FUNCTION_BLOCK FB_MachineController
VAR
	iConveyer : I_Conveyer;
	ePreviousMachineState : E_MachineState;
	fbTimer : TON;
	tWaitTime : TIME := T#10S;
	tProcessTime : TIME := T#5S;
	fbAutoTimer : TON;
END_VAR

IF GVL_HMI.bStop THEN
	IF GVL_HMI.eMachineState =  E_MachineState.STOPPED THEN
		GVL_HMI.eMachineState := E_MachineState.IDLE;
	ELSE
		ePreviousMachineState := GVL_HMI.eMachineState ;
		GVL_HMI.eMachineState := E_MachineState.STOPPED;
	END_IF
	fbTimer(IN := FALSE, PT := tWaitTime);
	GVL_HMI.bStop := FALSE;
	
END_IF
CASE GVL_HMI.eMachineState OF
	E_MachineState.IDLE :
		IF GVL_HMI.bStart THEN
			GVL_HMI.bStart := FALSE;
			IF iConveyer <> 0 THEN
					ePreviousMachineState := GVL_HMI.eMachineState ;
					GVL_HMI.eMachineState := E_MachineState.WAIT_FOR_BOTTLE;
			ELSE
				ePreviousMachineState := GVL_HMI.eMachineState ;
				GVL_HMI.eMachineState := E_MachineState.ERROR;
			END_IF
		END_IF
		
	E_MachineState.WAIT_FOR_BOTTLE :
		iConveyer.Start();
		fbTimer ( IN:= TRUE, PT:= tWaitTime);
		IF fbTimer.Q THEN
			fbTimer(IN := FALSE);
			GVL_HMI.eAlarmState := E_AlarmState.BOTTLE_SENSOR;
			GVL_HMI.eMachineState := E_MachineState.ERROR;
		END_IF
		//AutoMode
		IF GVL_HMI.eMachineMode = E_MachineMode.Auto THEN
			fbAutoTimer(IN := TRUE, PT := tProcessTime);
			IF fbAutoTimer.Q THEN
				fbAutoTimer(IN := FALSE);
				GVL_HMI.bBottleSensor := TRUE;
			END_IF
		ELSE
			fbAutoTimer(IN := FALSE);
		END_IF
		
		IF GVL_HMI.bBottleSensor THEN
				GVL_HMI.bBottleSensor := FALSE;
				fbTimer(IN := FALSE);
				iConveyer.Stop();
				ePreviousMachineState := GVL_HMI.eMachineState ;
				GVL_HMI.eMachineState := E_MachineState.FILLING;
		END_IF
	
	E_MachineState.FILLING :
		GVL_HMI.bFillingValve := TRUE;
		fbTimer ( IN:= TRUE, PT:= tWaitTime);
		IF fbTimer.Q THEN
			fbTimer(IN := FALSE);
			GVL_HMI.eAlarmState := E_AlarmState.LEVEL_SENSOR;
			GVL_HMI.eMachineState := E_MachineState.ERROR;
		END_IF
		//AutoMode
		IF GVL_HMI.eMachineMode = E_MachineMode.Auto THEN
			fbAutoTimer(IN := TRUE, PT := tProcessTime);
			IF fbAutoTimer.Q THEN
				fbAutoTimer(IN := FALSE);
				GVL_HMI.bLevelSensor := TRUE;
			END_IF
		ELSE
			fbAutoTimer(IN := FALSE);
		END_IF
		
		IF GVL_HMI.bLevelSensor THEN
				fbTimer(IN := FALSE);
				GVL_HMI.bFillingValve := FALSE;
				ePreviousMachineState := GVL_HMI.eMachineState ;
				GVL_HMI.eMachineState := E_MachineState.COMPLETED;
		END_IF
	
	E_MachineState.COMPLETED :
			GVL_HMI.bLevelSensor := FALSE;
			iConveyer.Start();
			GVL_HMI.bBottleSensor := FALSE;
			ePreviousMachineState := GVL_HMI.eMachineState ;
			
			//Auto
			IF GVL_HMI.eMachineMode = E_MachineMode.Auto THEN
				GVL_HMI.nBottleCounter := GVL_HMI.nBottleCounter + 1;
				GVL_HMI.eMachineState := E_MachineState.WAIT_FOR_BOTTLE;
				
			ELSE
				IF GVL_HMI.bStart THEN
					GVL_HMI.nBottleCounter := GVL_HMI.nBottleCounter + 1;
					GVL_HMI.bStart := FALSE;
					GVL_HMI.eMachineState := E_MachineState.WAIT_FOR_BOTTLE;
					
				END_IF
			END_IF
			
	
	E_MachineState.STOPPED :
			iConveyer.Stop();
			GVL_HMI.bFillingValve := FALSE;
			IF GVL_HMI.bStart THEN
				GVL_HMI.bStart := FALSE;
				GVL_HMI.eMachineState := ePreviousMachineState;
			END_IF
	E_MachineState.ERROR :
		iConveyer.Stop();
		GVL_HMI.bFillingValve := FALSE;
		IF GVL_HMI.bReset THEN
			GVL_HMI.bBottleSensor := FALSE;
			GVL_HMI.bLevelSensor := FALSE;
			GVL_HMI.bReset := FALSE;
			GVL_HMI.bAlarmLamp := FALSE;
			GVL_HMI.eAlarmState := E_AlarmState.OFF;
			GVL_HMI.eMachineState := E_MachineState.IDLE;
		END_IF
END_CASE

METHOD FB_init : BOOL
VAR_INPUT
	bInitRetains : BOOL; // if TRUE, the retain variables are initialized (warm start / cold start)
	bInCopyCode : BOOL;  // if TRUE, the instance afterwards gets moved into the copy code (online change)
	_iConveyer : I_Conveyer;
END_VAR
iConveyer := _iConveyer;
END_METHOD

END_FUNCTION_BLOCK

(* stored: Version 1.1.0.1, ProductVersion 3.1.4024.16
   POU FB_MachineController: Id {ef67becc-e70d-412b-b4ad-4db246967a51}, SpecialFunc None
   Method FB_init: Id {87659227-88b5-4fb8-8a31-a04d98ebd634} *)
